// TIA Portal V20 export
TYPE "type_emRelations_em2_jobInterface"
// stored: Access Published, Namespace Unit1
   STRUCT
      requset : Struct
         reqUnwinderTopReWind : Bool;
         reqUnwinderBtmReWind : Bool;
         reqEm0To1LinkChg : Bool;
         reqEm1To0LinkChg : Bool;
         reqDancerOn : Bool;
         reqDancerOff : Bool;
      END_STRUCT;
      ready : Struct
         null : Bool;
      END_STRUCT;
      busy : Struct
         busyAutoSplice : Bool;
      END_STRUCT;
      done : Struct
         doneAutoSplice : Bool;
      END_STRUCT;
      workingDone : Struct
         homeJob1WorkingDone { S7_SetPoint := 'True'} : Bool;
         suctionPadUpJob2WorkingDone : Bool;
         topSepaVaccumJob3WorkingDone : Bool;
         btmSepaVaccumJob4WorkingDone : Bool;
         cuttingJob5WorkingDone : Bool;
         topSepaTransferJob6WorkingDone : Bool;
         btmSepaTransferJob7WorkingDone : Bool;
         suctionPadDownJob8WorkingDone : Bool;
         topSepaReMoveJob9WorkingDone : Bool;
         btmSepaReMoveJob10WorkingDone : Bool;
         topSpliceRoateJob11WorkingDone : Bool;
         btmSpliceRoateJob12WorkingDone : Bool;
         topTapingStartJob13WorkingDone : Bool;
         btmTapingStartJob14WorkingDone : Bool;
         tapingFinishJob15WorkingDone : Bool;
         fullAutoSplicingJob30WorkingDone : Bool;
      END_STRUCT;
   END_STRUCT;
END_TYPE
